TYPE ST_Diagnostic :
STRUCT
	Temperature			:UDINT;
	BootCount			:UDINT;
	OperationTime		:UDINT;
	OperationDuration	:ARRAY[0..2] OF INT;
END_STRUCT
END_TYPE

(* stored: Version 1.1.0.1, ProductVersion 3.1.4024.12
   DUT ST_Diagnostic: Id {654957b3-4771-4c01-a6c2-f95c529c28fc} *)
